FUNCTION_BLOCK FB_MafacJava
VAR_INPUT
END_VAR
VAR_OUTPUT
END_VAR
VAR
END_VAR

END_FUNCTION_BLOCK

(* stored: Version 1.1.0.1, ProductVersion 3.1.4024.10
   POU FB_MafacJava: Id {9ab89f15-d411-40eb-9781-2f3a2eb9a02c}, SpecialFunc None *)
